// TIA Portal V20 export
FUNCTION "ManOperationCm_typeAxisControlInterface" : Void   // FC76, LAD
// stored: SetENOAutomatically false
   VAR_INPUT
      disableUnit : Bool;
   END_VAR
   VAR_OUTPUT
      Status : Word;
      errorID : Word;
   END_VAR
   VAR_IN_OUT
      manualOperationEm : "LAF_typeManEm";
      manualOperationEmArea : "LAF_typeManOperationArea";
      manualOperationCms : "LAF_typeManOperation";
      Axis : "LBC_typeAxisControlInterface";
   END_VAR
BEGIN

REGION Network 1: Manual Operation Cm - typeAxisControlInterface
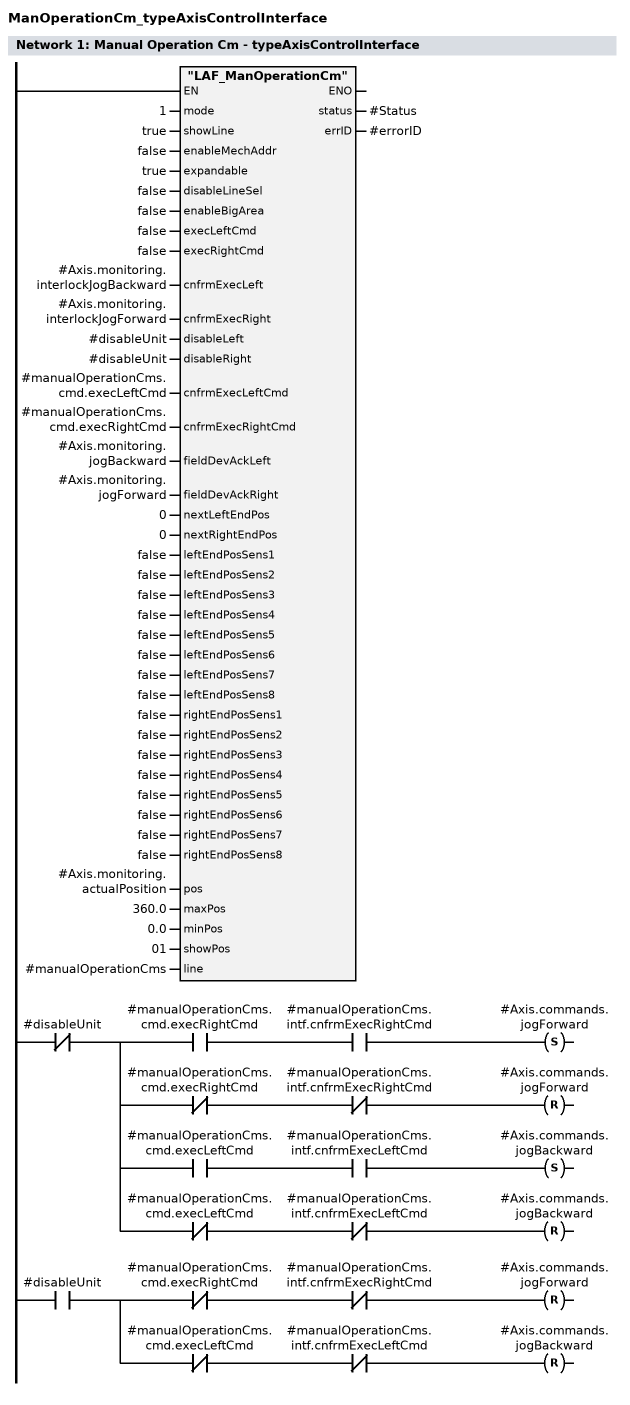
   RUNG wire#powerrail
      "LAF_ManOperationCm"(mode := 1, showLine := true, enableMechAddr := false, expandable := true, disableLineSel := false, enableBigArea := false, execLeftCmd := false, execRightCmd := false, cnfrmExecLeft := #Axis.monitoring.interlockJogBackward, cnfrmExecRight := #Axis.monitoring.interlockJogForward, disableLeft := #disableUnit, disableRight := #disableUnit, cnfrmExecLeftCmd := #manualOperationCms.cmd.execLeftCmd, cnfrmExecRightCmd := #manualOperationCms.cmd.execRightCmd, fieldDevAckLeft := #Axis.monitoring.jogBackward, fieldDevAckRight := #Axis.monitoring.jogForward, nextLeftEndPos := 0, nextRightEndPos := 0, leftEndPosSens1 := false, leftEndPosSens2 := false, leftEndPosSens3 := false, leftEndPosSens4 := false, leftEndPosSens5 := false, leftEndPosSens6 := false, leftEndPosSens7 := false, leftEndPosSens8 := false, rightEndPosSens1 := false, rightEndPosSens2 := false, rightEndPosSens3 := false, rightEndPosSens4 := false, rightEndPosSens5 := false, rightEndPosSens6 := false, rightEndPosSens7 := false, rightEndPosSens8 := false, pos := #Axis.monitoring.actualPosition, maxPos := 360.0, minPos := 0.0, showPos := 01, line := #manualOperationCms, status => #Status, errID => #errorID)
   END_RUNG
   RUNG wire#powerrail
      I_Contact( #disableUnit )
      wire#w1
      Contact( #manualOperationCms.cmd.execRightCmd )
      Contact( #manualOperationCms.intf.cnfrmExecRightCmd )
      S_Coil( #Axis.commands.jogForward )
   END_RUNG
   RUNG wire#w1
      I_Contact( #manualOperationCms.cmd.execRightCmd )
      I_Contact( #manualOperationCms.intf.cnfrmExecRightCmd )
      R_Coil( #Axis.commands.jogForward )
   END_RUNG
   RUNG wire#w1
      Contact( #manualOperationCms.cmd.execLeftCmd )
      Contact( #manualOperationCms.intf.cnfrmExecLeftCmd )
      S_Coil( #Axis.commands.jogBackward )
   END_RUNG
   RUNG wire#w1
      I_Contact( #manualOperationCms.cmd.execLeftCmd )
      I_Contact( #manualOperationCms.intf.cnfrmExecLeftCmd )
      R_Coil( #Axis.commands.jogBackward )
   END_RUNG
   RUNG wire#powerrail
      Contact( #disableUnit )
      wire#w2
      I_Contact( #manualOperationCms.cmd.execRightCmd )
      I_Contact( #manualOperationCms.intf.cnfrmExecRightCmd )
      R_Coil( #Axis.commands.jogForward )
   END_RUNG
   RUNG wire#w2
      I_Contact( #manualOperationCms.cmd.execLeftCmd )
      I_Contact( #manualOperationCms.intf.cnfrmExecLeftCmd )
      R_Coil( #Axis.commands.jogBackward )
   END_RUNG
   // the same network as SCL:
   "LAF_ManOperationCm"(mode := 1,
                        showLine := true,
                        enableMechAddr := false,
                        expandable := true,
                        disableLineSel := false,
                        enableBigArea := false,
                        execLeftCmd := false,
                        execRightCmd := false,
                        cnfrmExecLeft := #Axis.monitoring.interlockJogBackward,
                        cnfrmExecRight := #Axis.monitoring.interlockJogForward,
                        disableLeft := #disableUnit,
                        disableRight := #disableUnit,
                        cnfrmExecLeftCmd := #manualOperationCms.cmd.execLeftCmd,
                        cnfrmExecRightCmd := #manualOperationCms.cmd.execRightCmd,
                        fieldDevAckLeft := #Axis.monitoring.jogBackward,
                        fieldDevAckRight := #Axis.monitoring.jogForward,
                        nextLeftEndPos := 0,
                        nextRightEndPos := 0,
                        leftEndPosSens1 := false,
                        leftEndPosSens2 := false,
                        leftEndPosSens3 := false,
                        leftEndPosSens4 := false,
                        leftEndPosSens5 := false,
                        leftEndPosSens6 := false,
                        leftEndPosSens7 := false,
                        leftEndPosSens8 := false,
                        rightEndPosSens1 := false,
                        rightEndPosSens2 := false,
                        rightEndPosSens3 := false,
                        rightEndPosSens4 := false,
                        rightEndPosSens5 := false,
                        rightEndPosSens6 := false,
                        rightEndPosSens7 := false,
                        rightEndPosSens8 := false,
                        pos := #Axis.monitoring.actualPosition,
                        maxPos := 360.0,
                        minPos := 0.0,
                        showPos := 01,
                        line := #manualOperationCms,
                        status => #Status,
                        errID => #errorID);
   IF NOT #disableUnit AND #manualOperationCms.cmd.execRightCmd AND #manualOperationCms.intf.cnfrmExecRightCmd THEN
       #Axis.commands.jogForward := TRUE;
   END_IF;
   IF NOT #disableUnit AND NOT #manualOperationCms.cmd.execRightCmd AND NOT #manualOperationCms.intf.cnfrmExecRightCmd THEN
       #Axis.commands.jogForward := FALSE;
   END_IF;
   IF NOT #disableUnit AND #manualOperationCms.cmd.execLeftCmd AND #manualOperationCms.intf.cnfrmExecLeftCmd THEN
       #Axis.commands.jogBackward := TRUE;
   END_IF;
   IF NOT #disableUnit AND NOT #manualOperationCms.cmd.execLeftCmd AND NOT #manualOperationCms.intf.cnfrmExecLeftCmd THEN
       #Axis.commands.jogBackward := FALSE;
   END_IF;
   IF #disableUnit AND NOT #manualOperationCms.cmd.execRightCmd AND NOT #manualOperationCms.intf.cnfrmExecRightCmd THEN
       #Axis.commands.jogForward := FALSE;
   END_IF;
   IF #disableUnit AND NOT #manualOperationCms.cmd.execLeftCmd AND NOT #manualOperationCms.intf.cnfrmExecLeftCmd THEN
       #Axis.commands.jogBackward := FALSE;
   END_IF;
END_REGION
END_FUNCTION
